// TIA Portal V17 export
// export: Created 2024-08-09T12:53:12.848557Z, ExportSetting WithDefaults, DisplayName Totally Integrated Automation Portal, DisplayVersion V17 Update 7, DisplayName TIA Portal Openness, DisplayVersion V17 Update 7, DisplayName TIA Portal Version Control Interface, DisplayVersion V17, DisplayName STEP 7 Professional, DisplayVersion V17 Update 7, DisplayName STEP 7 Safety, DisplayVersion V17 Update 6, DisplayName WinCC Professional, DisplayVersion V17 Update 7
VAR_GLOBAL   // PLC tag table "SurvDosBenne"
END_VAR
VAR_GLOBAL CONSTANT   // user constants
   NIV_SURDOS_DEBUT_LOT : USInt := 1;
   NIV_SURDOS_ATT_FIN_DOSAGE : USInt := 10;
   NIV_SURDOS_FIN_DOSAGE_PES_PARTIELLE : USInt := 20;
   NIV_SURDOS_VIDANGE_PES_PARTIELLE : USInt := 40;
   NIV_SURDOS_VID_PARTIELLE_DEPUIS_X_SEC : USInt := 41;
   NIV_SURDOS_FIN_VIDANGE_PES_PARTIELLE : USInt := 43;
   NIV_SURDOS_FIN_DOSAGE_DERNIERE_PESEE : USInt := 50;
   NIV_SURDOS_FIN_DOSAGE_AVEC_PRODUIT : USInt := 55;
   NIV_SURDOS_ATT_FIN_REMPLISSAGE : USInt := 57;
   NIV_SURDOS_DEBUT_VIDANGE_BENNE : USInt := 60;
   NIV_SURDOS_VID_DEPUIS_X_SEC : USInt := 62;
   NIV_SURDOS_ARRET_VIDANGE_BENNE : USInt := 65;
   NIV_SURDOS_BENNE_VIDE : USInt := 70;
   NIV_SURDOS_FIN_VIDANGE_BENNE : USInt := 80;
   NIV_SURDOS_FIN_LOT : USInt := 255;
END_VAR
